// TIA Portal project "Project1" (V19)

(* hardware
DEVICE "S7-1500/ET200MP station_1"  S7-1500 station
   slot 0: "Rail_0"  Rack  6ES7 590-1***0-0AA0
   slot 1: "PLC_1"  CPU 1513-1 PN  6ES7 513-1AL02-0AB0  V2.9
      slot 3: "CPU display_1"  6ES7591-1AA00-0AA0
      slot 32768: "PROFINET interface_1"  X1
         slot 32769: "Port_1"  X1 P1
         slot 32770: "Port_2"  X1 P2
      slot 34817: "Virtual CP interface port_1"  Virtual CP interface port  Virtual CP interface port
   slot 2: "DI 16x24VDC BA_1"  DI 16x24VDC BA  6ES7 521-1BH10-0AA0  V1.1
   slot 3: "DQ 16x24VDC/0.5A BA_1"  DQ 16x24VDC/0.5A BA  6ES7 522-1BH10-0AA0  V1.1
DEVICE "HMI_1"  KTP700 Basic PN
   slot 0: "HMI_1"  KTP700 Basic PN  6AV2 123-2GB03-0AX0  17.0.0.0
   slot 1: "HMI_RT_1"  KTP700 Basic PN  6AV2 123-2GB03-0AX0  17.0.0.0
   slot 5: "HMI_1.IE_CP_1"  PROFINET Interface  17.0.0.0
      slot 1: "PROFINET Interface_1"  PROFINET Interface
         slot 1: "Port_1"  Port
*)

// ===== PLC "PLC_1"  CPU 1513-1 PN =====

VAR_GLOBAL   // PLC tag table "Default tag table"
   "At Entry" AT %I0.0 : Bool;
   "At Load" AT %I0.1 : Bool;
   "At left" AT %I0.2 : Bool;
   "At Middle" AT %I0.3 : Bool;
   "At Right" AT %I0.4 : Bool;
   "At Unload" AT %I0.5 : Bool;
   "At Exit" AT %I0.6 : Bool;
   "Moving X" AT %I0.7 : Bool;
   "Moving Z" AT %I1.0 : Bool;
   "Start" AT %M3.1 : Bool;
   "Reset" AT %I1.2 : Bool;
   "Stop" AT %M3.3 : Bool;
   "Emergency stop" AT %I1.4 : Bool;
   "Auto" AT %I1.5 : Bool;
   "FACTORY I/O (Runing)" AT %I1.6 : Bool;
   "Entry Conveyor" AT %Q0.0 : Bool;
   "Load Conveyor" AT %Q0.1 : Bool;
   "Forks Left" AT %Q0.2 : Bool;
   "Forks Right" AT %Q0.3 : Bool;
   "Lift" AT %Q0.4 : Bool;
   "Unload Conveyor" AT %Q0.5 : Bool;
   "Exit Conveyor" AT %Q0.6 : Bool;
   "Start light" AT %Q0.7 : Bool;
   "Reset light" AT %Q1.0 : Bool;
   "Stop light" AT %Q1.1 : Bool;
   "Target position" AT %QW30 : Int;
   "State0" AT %M0.0 : Bool;
   "State1" AT %M0.1 : Bool;
   "State2" AT %M0.2 : Bool;
   "State3" AT %M0.3 : Bool;
   "State4" AT %M0.4 : Bool;
   "State5" AT %M0.5 : Bool;
   "State6" AT %M0.6 : Bool;
   "State7" AT %M0.7 : Bool;
   "State8" AT %M1.0 : Bool;
   "State9" AT %M1.1 : Bool;
   "Tag_1" AT %M1.3 : Bool;
   "Tag_2" AT %M1.4 : Bool;
   "Tag_3" AT %M1.5 : Bool;
   "Tag_4" AT %M1.6 : Bool;
   "Tag_5" AT %M1.2 : Bool;
   "t" AT %MW30 : Int;
   "Tag_6" AT %M1.7 : Bool;
END_VAR

FUNCTION "start stop" : Void   // FC1, LAD
{ S7_Optimized_Access := 'FALSE' }
VERSION : 0.1
BEGIN

REGION Network 1
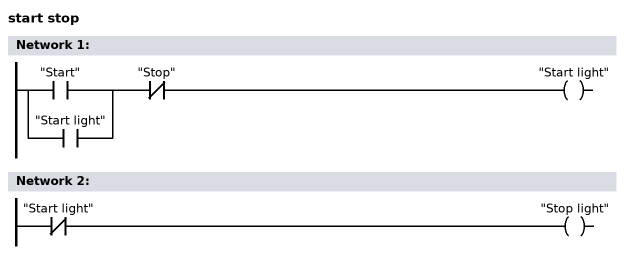
   RUNG wire#powerrail
      Contact( "Start" )
      wire#w1
      I_Contact( "Stop" )
      Coil( "Start light" )
   END_RUNG
   RUNG wire#powerrail
      Contact( "Start light" )
   END_RUNG wire#w1
   // the same network as SCL:
   "Start light" := ("Start" OR "Start light") AND NOT "Stop";
END_REGION

REGION Network 2
   RUNG wire#powerrail
      I_Contact( "Start light" )
      Coil( "Stop light" )
   END_RUNG
   // the same network as SCL:
   "Stop light" := NOT "Start light";
END_REGION
END_FUNCTION

FUNCTION "states" : Void   // FC2, LAD
{ S7_Optimized_Access := 'FALSE' }
VERSION : 0.1
   VAR_TEMP   // added for the SCL form of the ladder/FBD networks
      _w1 : Bool;
      _w2 : Bool;
   END_VAR
BEGIN

REGION Network 1
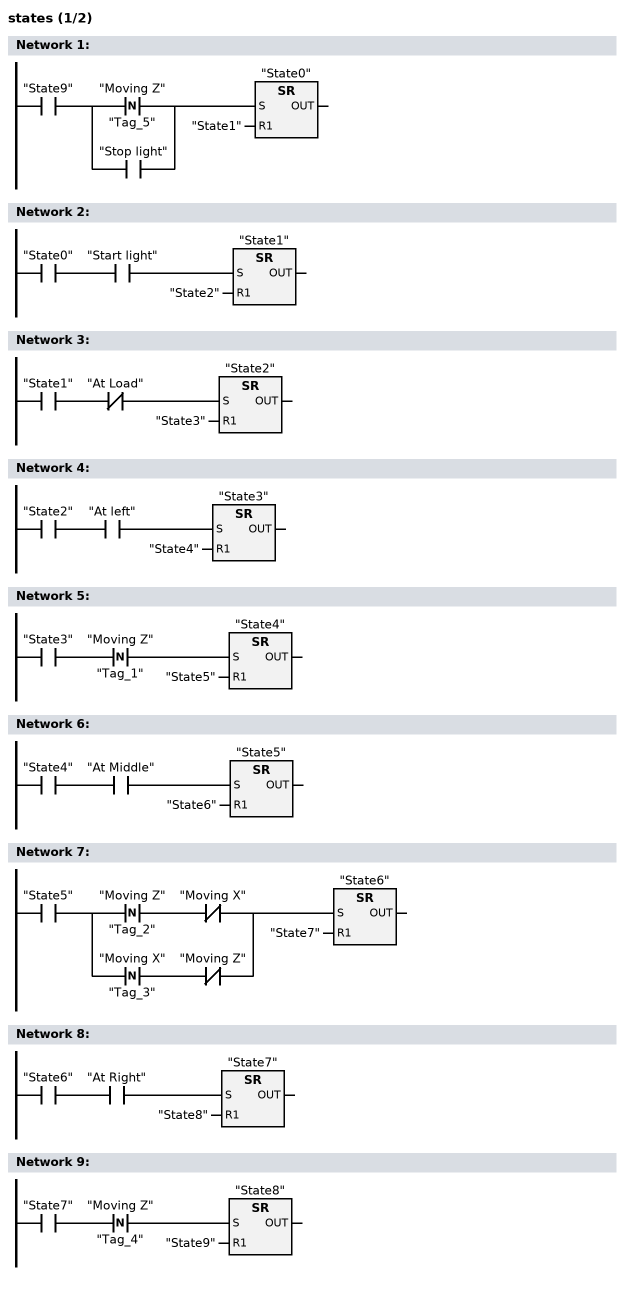
   RUNG wire#powerrail
      Contact( "State9" )
      wire#w1
      N_Contact(operand := "Moving Z", bit := "Tag_5")
      wire#w2
      S_SR(operand := "State0", r1 := "State1")
   END_RUNG
   RUNG wire#w1
      Contact( "Stop light" )
   END_RUNG wire#w2
   // the same network as SCL:
   #_w1 := "State9" AND NOT "Moving Z" AND "Tag_5";   // falling edge of "Moving Z"
   "Tag_5" := "Moving Z";
   IF #_w1 OR ("State9" AND "Stop light") THEN
       "State0" := TRUE;   // SR flip-flop
   END_IF;
   IF "State1" THEN "State0" := FALSE; END_IF;
END_REGION

REGION Network 2
   RUNG wire#powerrail
      Contact( "State0" )
      Contact( "Start light" )
      S_SR(operand := "State1", r1 := "State2")
   END_RUNG
   // the same network as SCL:
   IF "State0" AND "Start light" THEN
       "State1" := TRUE;   // SR flip-flop
   END_IF;
   IF "State2" THEN "State1" := FALSE; END_IF;
END_REGION

REGION Network 3
   RUNG wire#powerrail
      Contact( "State1" )
      I_Contact( "At Load" )
      S_SR(operand := "State2", r1 := "State3")
   END_RUNG
   // the same network as SCL:
   IF "State1" AND NOT "At Load" THEN
       "State2" := TRUE;   // SR flip-flop
   END_IF;
   IF "State3" THEN "State2" := FALSE; END_IF;
END_REGION

REGION Network 4
   RUNG wire#powerrail
      Contact( "State2" )
      Contact( "At left" )
      S_SR(operand := "State3", r1 := "State4")
   END_RUNG
   // the same network as SCL:
   IF "State2" AND "At left" THEN
       "State3" := TRUE;   // SR flip-flop
   END_IF;
   IF "State4" THEN "State3" := FALSE; END_IF;
END_REGION

REGION Network 5
   RUNG wire#powerrail
      Contact( "State3" )
      N_Contact(operand := "Moving Z", bit := "Tag_1")
      S_SR(operand := "State4", r1 := "State5")
   END_RUNG
   // the same network as SCL:
   #_w1 := "State3" AND NOT "Moving Z" AND "Tag_1";   // falling edge of "Moving Z"
   "Tag_1" := "Moving Z";
   IF #_w1 THEN
       "State4" := TRUE;   // SR flip-flop
   END_IF;
   IF "State5" THEN "State4" := FALSE; END_IF;
END_REGION

REGION Network 6
   RUNG wire#powerrail
      Contact( "State4" )
      Contact( "At Middle" )
      S_SR(operand := "State5", r1 := "State6")
   END_RUNG
   // the same network as SCL:
   IF "State4" AND "At Middle" THEN
       "State5" := TRUE;   // SR flip-flop
   END_IF;
   IF "State6" THEN "State5" := FALSE; END_IF;
END_REGION

REGION Network 7
   RUNG wire#powerrail
      Contact( "State5" )
      wire#w1
      N_Contact(operand := "Moving Z", bit := "Tag_2")
      I_Contact( "Moving X" )
      wire#w2
      S_SR(operand := "State6", r1 := "State7")
   END_RUNG
   RUNG wire#w1
      N_Contact(operand := "Moving X", bit := "Tag_3")
      I_Contact( "Moving Z" )
   END_RUNG wire#w2
   // the same network as SCL:
   #_w1 := "State5" AND NOT "Moving Z" AND "Tag_2";   // falling edge of "Moving Z"
   "Tag_2" := "Moving Z";
   #_w2 := "State5" AND NOT "Moving X" AND "Tag_3";   // falling edge of "Moving X"
   "Tag_3" := "Moving X";
   IF (#_w1 AND NOT "Moving X") OR (#_w2 AND NOT "Moving Z") THEN
       "State6" := TRUE;   // SR flip-flop
   END_IF;
   IF "State7" THEN "State6" := FALSE; END_IF;
END_REGION

REGION Network 8
   RUNG wire#powerrail
      Contact( "State6" )
      Contact( "At Right" )
      S_SR(operand := "State7", r1 := "State8")
   END_RUNG
   // the same network as SCL:
   IF "State6" AND "At Right" THEN
       "State7" := TRUE;   // SR flip-flop
   END_IF;
   IF "State8" THEN "State7" := FALSE; END_IF;
END_REGION

REGION Network 9
   RUNG wire#powerrail
      Contact( "State7" )
      N_Contact(operand := "Moving Z", bit := "Tag_4")
      S_SR(operand := "State8", r1 := "State9")
   END_RUNG
   // the same network as SCL:
   #_w1 := "State7" AND NOT "Moving Z" AND "Tag_4";   // falling edge of "Moving Z"
   "Tag_4" := "Moving Z";
   IF #_w1 THEN
       "State8" := TRUE;   // SR flip-flop
   END_IF;
   IF "State9" THEN "State8" := FALSE; END_IF;
END_REGION

REGION Network 10
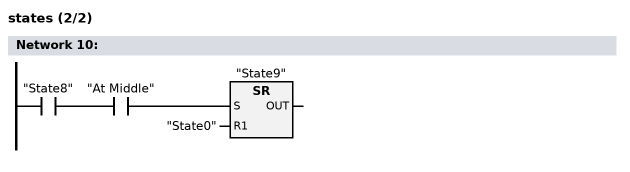
   RUNG wire#powerrail
      Contact( "State8" )
      Contact( "At Middle" )
      S_SR(operand := "State9", r1 := "State0")
   END_RUNG
   // the same network as SCL:
   IF "State8" AND "At Middle" THEN
       "State9" := TRUE;   // SR flip-flop
   END_IF;
   IF "State0" THEN "State9" := FALSE; END_IF;
END_REGION
END_FUNCTION

FUNCTION "actuators" : Void   // FC3, LAD
{ S7_Optimized_Access := 'FALSE' }
VERSION : 0.1
   VAR_TEMP   // added for the SCL form of the ladder/FBD networks
      _w1 : Bool;
   END_VAR
BEGIN

REGION Network 1
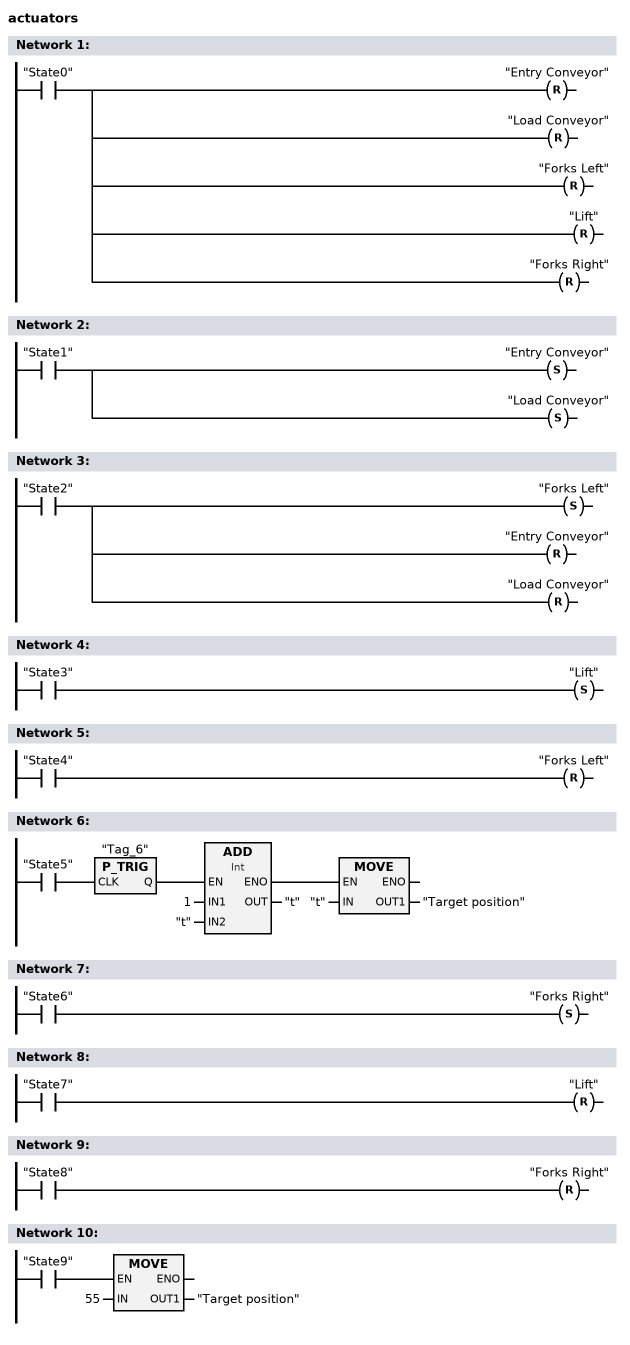
   RUNG wire#powerrail
      Contact( "State0" )
      wire#w1
      R_Coil( "Entry Conveyor" )
   END_RUNG
   RUNG wire#w1
      R_Coil( "Load Conveyor" )
   END_RUNG
   RUNG wire#w1
      R_Coil( "Forks Left" )
   END_RUNG
   RUNG wire#w1
      R_Coil( "Lift" )
   END_RUNG
   RUNG wire#w1
      R_Coil( "Forks Right" )
   END_RUNG
   // the same network as SCL:
   IF "State0" THEN
       "Entry Conveyor" := FALSE;
       "Load Conveyor" := FALSE;
       "Forks Left" := FALSE;
       "Lift" := FALSE;
       "Forks Right" := FALSE;
   END_IF;
END_REGION

REGION Network 2
   RUNG wire#powerrail
      Contact( "State1" )
      wire#w1
      S_Coil( "Entry Conveyor" )
   END_RUNG
   RUNG wire#w1
      S_Coil( "Load Conveyor" )
   END_RUNG
   // the same network as SCL:
   IF "State1" THEN
       "Entry Conveyor" := TRUE;
       "Load Conveyor" := TRUE;
   END_IF;
END_REGION

REGION Network 3
   RUNG wire#powerrail
      Contact( "State2" )
      wire#w1
      S_Coil( "Forks Left" )
   END_RUNG
   RUNG wire#w1
      R_Coil( "Entry Conveyor" )
   END_RUNG
   RUNG wire#w1
      R_Coil( "Load Conveyor" )
   END_RUNG
   // the same network as SCL:
   IF "State2" THEN
       "Forks Left" := TRUE;
       "Entry Conveyor" := FALSE;
       "Load Conveyor" := FALSE;
   END_IF;
END_REGION

REGION Network 4
   RUNG wire#powerrail
      Contact( "State3" )
      S_Coil( "Lift" )
   END_RUNG
   // the same network as SCL:
   IF "State3" THEN "Lift" := TRUE; END_IF;
END_REGION

REGION Network 5
   RUNG wire#powerrail
      Contact( "State4" )
      R_Coil( "Forks Left" )
   END_RUNG
   // the same network as SCL:
   IF "State4" THEN "Forks Left" := FALSE; END_IF;
END_REGION

REGION Network 6
   RUNG wire#powerrail
      Contact( "State5" )
      P_Trig( "Tag_6" )
      { S7_Templates := "SrcType := Int"; S7_GenerateENO := "TRUE" } Add(in1 := 1, in2 := "t", out => "t")
      { S7_GenerateENO := "TRUE" } Move(in := "t", out1 => "Target position")
   END_RUNG
   // the same network as SCL:
   // ENO of a box is taken as its EN; it also drops when the box reports an error
   #_w1 := "State5" AND NOT "Tag_6";   // rising edge
   "Tag_6" := "State5";
   IF #_w1 THEN
       "t" := 1 + "t";
       "Target position" := "t";
   END_IF;
END_REGION

REGION Network 7
   RUNG wire#powerrail
      Contact( "State6" )
      S_Coil( "Forks Right" )
   END_RUNG
   // the same network as SCL:
   IF "State6" THEN "Forks Right" := TRUE; END_IF;
END_REGION

REGION Network 8
   RUNG wire#powerrail
      Contact( "State7" )
      R_Coil( "Lift" )
   END_RUNG
   // the same network as SCL:
   IF "State7" THEN "Lift" := FALSE; END_IF;
END_REGION

REGION Network 9
   RUNG wire#powerrail
      Contact( "State8" )
      R_Coil( "Forks Right" )
   END_RUNG
   // the same network as SCL:
   IF "State8" THEN "Forks Right" := FALSE; END_IF;
END_REGION

REGION Network 10
   RUNG wire#powerrail
      Contact( "State9" )
      { S7_GenerateENO := "TRUE" } Move(in := 55, out1 => "Target position")
   END_RUNG
   // the same network as SCL:
   IF "State9" THEN "Target position" := 55; END_IF;
END_REGION
END_FUNCTION

ORGANIZATION_BLOCK "Main"   // OB1, LAD, ProgramCycle
TITLE = "Main Program Sweep (Cycle)"
{ S7_Optimized_Access := 'FALSE' }
VERSION : 0.1
   VAR_TEMP
      OB1_EV_CLASS : Byte;   // Bits 0-3 = 1 (Coming event), Bits 4-7 = 1 (Event class 1)
      OB1_SCAN_1 : Byte;   // 1 (Cold restart scan 1 of OB 1), 3 (Scan 2-n of OB 1)
      OB1_PRIORITY : Byte;   // Priority of OB Execution
      OB1_OB_NUMBR : Byte;   // 1 (Organization block 1, OB1)
      OB1_RESERVED_1 : Byte;   // Reserved for system
      OB1_RESERVED_2 : Byte;   // Reserved for system
      OB1_PREV_CYCLE : Int;   // Cycle time of previous OB1 scan (milliseconds)
      OB1_MIN_CYCLE : Int;   // Minimum cycle time of OB1 (milliseconds)
      OB1_MAX_CYCLE : Int;   // Maximum cycle time of OB1 (milliseconds)
      OB1_DATE_TIME : Date_And_Time;   // Date and time OB1 started
   END_VAR
BEGIN

REGION Network 1
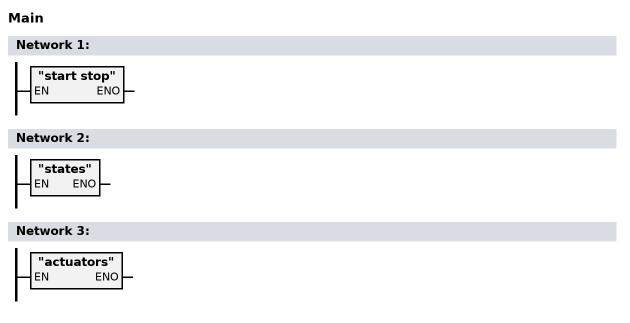
   RUNG wire#powerrail
      "start stop"()
   END_RUNG
   // the same network as SCL:
   "start stop"();
END_REGION

REGION Network 2
   RUNG wire#powerrail
      "states"()
   END_RUNG
   // the same network as SCL:
   "states"();
END_REGION

REGION Network 3
   RUNG wire#powerrail
      "actuators"()
   END_RUNG
   // the same network as SCL:
   "actuators"();
END_REGION
END_ORGANIZATION_BLOCK

ORGANIZATION_BLOCK "COMPLETE RESTART"   // OB100, LAD, Startup
TITLE = "Complete Restart"
{ S7_Optimized_Access := 'FALSE' }
VERSION : 0.1
   VAR_TEMP
      OB100_EV_CLASS : Byte;   // 16#13, Event class 1, Entering event state, Event logged in diagnostic buffer
      OB100_STRTUP : Byte;   // 16#81/82/83/84 Method of startup
      OB100_PRIORITY : Byte;   // Priority of OB Execution
      OB100_OB_NUMBR : Byte;   // 100 (Organization block 100, OB100)
      OB100_RESERVED_1 : Byte;   // Reserved for system
      OB100_RESERVED_2 : Byte;   // Reserved for system
      OB100_STOP : Word;   // Event that caused CPU to stop (16#4xxx)
      OB100_STRT_INFO : DWord;   // Information on how system started
      OB100_DATE_TIME : Date_And_Time;   // Date and time OB100 started
   END_VAR
BEGIN

REGION Network 1
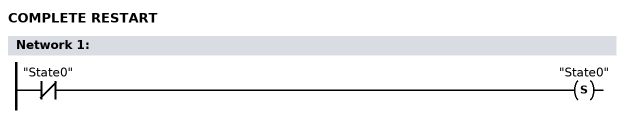
   RUNG wire#powerrail
      I_Contact( "State0" )
      S_Coil( "State0" )
   END_RUNG
   // the same network as SCL:
   IF NOT "State0" THEN "State0" := TRUE; END_IF;
END_REGION
END_ORGANIZATION_BLOCK

(* ===== HMI "HMI_RT_1" =====
system functions are stored by id; their names below are inferred from use
connection "HMI_Connection_1": ETHERNET, SMART_S7_1500_OMS

HMI tags "Default tag table"
   "Tag_ScreenNumber" : UInt, internal
   "Start light" : Bool = PLC "Start light" AT %Q0.7, 1 s
   "Start" : Bool = PLC Start AT %M3.1, 1 s
   "Stop" : Bool = PLC Stop AT %M3.3, 1 s
   "t" : Int = PLC t AT %MW30, 1 s

Template "Template_1" 800x480
   Button "Exit" at 714,429 size 71x50; TextOff 'Exit'; PictureOff "ExitRuntime_KTP700_Basic_PN_TR"; PictureOn "ExitRuntime_KTP700_Basic_PN_TR"
      on Release: StopRuntime(0)
   Button "Template_Button" at 614,429 size 71x50; TextOff 'Text'
   Button "Template_Button_1" at 514,429 size 71x50; TextOff 'Text'
   Button "Template_Button_2" at 414,429 size 71x50; TextOff 'Text'
   Button "Template_Button_3" at 314,429 size 71x50; TextOff 'Text'
   Button "Template_Button_4" at 214,429 size 71x50; TextOff 'Text'
   Button "Alarms" at 114,429 size 71x50; TextOff 'Alarms'; PictureOff "AlarmDisplay_KTP700_Basic_PN_TR"; PictureOn "AlarmDisplay_KTP700_Basic_PN_TR"
      on Release: function_ef3f5d25("Alarm window_Unacknowledged", -1)
   Button "Start screen" at 14,429 size 71x50; TextOff 'Start screen'; PictureOff "NavigateHome_KTP700_Basic_PN_TR"; PictureOn "NavigateHome_KTP700_Basic_PN_TR"
      on Release: ActivateScreen("Root screen", 0)
   SymbolicIOField "Symbolic_IO_Field_Screen" at 93,9 size 600x33; TextOff '0'; TextOn '1'; TextList "TextList_ScreenNames"
      ProcessValue <- "Tag_ScreenNumber"
      on Change: ActivateScreenByNumber("Tag_ScreenNumber", 0)
   DateTimeField "HmiScreenItemData" at 695,25 size 105x25
   DateTimeField "HmiScreenItemData_1" at 695,0 size 105x25
   GraphicView "Logo" at 0,0 size 91x51; Picture "Logo of HMI_1"

screen "Root screen" 800x480, template "Template_1"
   on GenerateScreen: SetTag("Tag_ScreenNumber", 1)
   TextField "HmiScreenItemData" at 80,225 size 640x25; Text 'Automated Warehouse'
   Button "Button_2" at 423,274 size 192x32; TextOff 'Automatic'; TextOn 'Screen_1'
      on Click: ActivateScreen("Screen_1", 0)
   Button "Button_3" at 182,274 size 192x32; TextOff 'Manual'; TextOn 'Screen_1'

screen "Screen_1" 800x480
   Button "Button_1" at 206,168 size 96x32; TextOff 'Start'
      on Click: SetBit("Start"); ResetBit("Stop")
   Button "Button_2" at 206,257 size 96x32; TextOff 'Stop'
      on Click: SetBit("Stop"); ResetBit("Start")
   Rectangle "Rectangle_1" at 422,168 size 96x48
      Appearance <- "Start light"
   IOField "I/O field_1" at 422,257 size 94x77; FormatPattern 9999999
      ProcessValue <- "t"
   Button "Button_3" at 1,445 size 192x32; TextOff 'Root screen'
      on Click: ActivateScreen("Root screen", 0)
*)